FUNCTION_BLOCK POU
VAR_INPUT
END_VAR
VAR_OUTPUT
END_VAR
VAR
END_VAR

// NETWORK 1

END_FUNCTION_BLOCK

(* stored: Version 1.1.0.1
   POU POU: Id {1bf8817e-3480-4905-ba78-895aabcbeb5c}, SpecialFunc None *)
